Yaskawa INFORM job: ROBOT.JBI

/JOB
//NAME ROBOT
//POS
///NPOS 25,0,0,0,0,0
///TOOL 0
///POSTYPE PULSE
///PULSE
C00000=-55572,28782,34434,-11577,-77346,20396
C00001=-66078,-29416,-50626,-80818,-25071,37969
C00002=-81236,73799,35237,-77959,-112523,43941
C00003=-32913,-25608,-44856,72411,-30097,-38142
C00004=-16277,56236,11362,72080,-101887,38552
C00005=-42062,-7834,-25997,-9399,-57401,15928
C00006=-18418,-2630,-27076,24974,-65995,50307
C00007=315,64603,-36897,85043,-114569,-52621
C00008=-53017,73506,38851,-20986,-116855,-38263
C00009=-74794,-25961,-78519,-90017,-54723,20981
C00010=-20365,-19310,-51345,-2901,-46047,4490
C00011=-62575,-2681,-78305,-82589,-71206,62019
C00012=-44317,-56748,-112019,-116729,-39654,94900
C00013=25617,53512,-59328,73700,-96599,15443
C00014=6004,76003,3668,32872,-115025,65194
C00015=69114,32290,-24931,-19486,-40863,30805
C00016=99031,92364,24408,42095,-89317,16855
C00017=57588,12307,-73691,-118107,-34600,84798
C00018=54063,105342,43343,-34503,-100414,-38145
C00019=72957,87992,41717,134,-88789,-29391
C00020=58027,-20436,-103590,-38607,-24469,49050
C00021=79265,61902,-40302,13716,-72208,-32504
C00022=46076,100212,-24560,-24651,-90441,2450
C00023=13173,73301,-84839,-72161,-75519,60290
C00024=15627,29677,-109648,-85880,-62831,91262
//INST
///DATE 2023/09/21 14:39
///ATTR SC,RW
///GROUP1 RB1
NOP
'*
MOVJ C00000 VJ=0.50 PL=8
MOVJ C00001 VJ=0.50 PL=8
MOVJ C00002 VJ=0.50 PL=8
MOVJ C00003 VJ=0.50 PL=8
MOVJ C00004 VJ=0.50 PL=8
'*
MOVJ C00005 VJ=0.50 PL=8
MOVJ C00006 VJ=0.50 PL=8
MOVJ C00007 VJ=0.50 PL=8
MOVJ C00008 VJ=0.50 PL=8
MOVJ C00009 VJ=0.50 PL=8
'*
MOVJ C00010 VJ=0.50 PL=8
MOVJ C00011 VJ=0.50 PL=8
MOVJ C00012 VJ=0.50 PL=8
MOVJ C00013 VJ=0.50 PL=8
MOVJ C00014 VJ=0.50 PL=8
'*
MOVJ C00015 VJ=0.50 PL=8
MOVJ C00016 VJ=0.50 PL=8
MOVJ C00017 VJ=0.50 PL=8
MOVJ C00018 VJ=0.50 PL=8
MOVJ C00019 VJ=0.50 PL=8
'*
MOVJ C00020 VJ=0.50 PL=8
MOVJ C00021 VJ=0.50 PL=8
MOVJ C00022 VJ=0.50 PL=8
MOVJ C00023 VJ=0.50 PL=8
MOVJ C00024 VJ=0.50 PL=8
END
